// TIA Portal V20 export
VAR_GLOBAL   // PLC tag table "TextListId"
END_VAR
VAR_GLOBAL CONSTANT   // user constants
   TEXT_LIST_ID_PN_DEV_DIAG : Int := 591;   // SICAR: ID of PLC Alarm text list
   TEXT_LIST_ID_CHECKSUM : Int := 584;   // SICAR: ID of PLC Alarm text list
   TEXT_LIST_ID_EEEMONITOR_REPORT : Int := 562;   // SICAR: ID of PLC Alarm text list
   TEXT_LIST_ID_EEEMONITOR_CALC : Int := 561;   // SICAR: ID of PLC Alarm text list
   TEXT_LIST_ID_IDENT_SYSTEM : Int := 516;   // SICAR: ID of PLC Alarm for ident demo
   TEXT_LIST_ID_SMC_PD : Int := 585;   // SICAR: ID of PLC Alarm text list
   TEXT_LIST_ID_MOTORSTARTERS : Int := 588;   // SICAR: ID of PLC Alarm for motorstarter Demo
   TEXT_LIST_ID_DEV_FWD_REV : Int := 592;   // SICAR: ID of PLC Alarm for motorstarter Demo
END_VAR
